// TIA Portal project "Lab3 with HMI" (V18)

(* hardware
DEVICE "HMI_1"  KTP700 Basic PN
   slot 0: "HMI_1"  KTP700 Basic PN  6AV2 123-2GB03-0AX0  15.1.0.0
   slot 1: "HMI_RT_1"  KTP700 Basic PN  6AV2 123-2GB03-0AX0  15.1.0.0
   slot 5: "HMI_1.IE_CP_1"  PROFINET Interface  15.0.1.0
      slot 1: "PROFINET Interface_1"  PROFINET Interface
         slot 1: "Port_1"  Port
DEVICE "S7-1200 station_1"  S7-1200 Station
   slot 0: "Rack_0"  S7-1200 Rack  Rack  V1.0
   slot 1: "PLC_1"  CPU 1214C DC/DC/DC  6ES7 214-1AG40-0XB0  V4.5
   slot 3: "ADC"  AQ1 signal board  6ES7 232-4HA30-0XB0  V1.0
DEVICE "S7-1200 station_2"  S7-1200 Station
   slot 0: "Rack_0"  S7-1200 Rack  Rack  V1.0
   slot 1: "PLC_2"  CPU 1215C DC/DC/DC  6ES7 215-1AG40-0XB0  V4.5
DEVICE "HMI_2"  KTP700 Basic PN
   slot 0: "HMI_2"  KTP700 Basic PN  6AV2 123-2GB03-0AX0  15.1.0.0
   slot 1: "HMI_RT_2"  KTP700 Basic PN  6AV2 123-2GB03-0AX0  15.1.0.0
   slot 5: "HMI_2.IE_CP_1"  PROFINET Interface  15.0.1.0
      slot 1: "PROFINET Interface_1"  PROFINET Interface
         slot 1: "Port_1"  Port
*)

// ===== PLC "PLC_1"  CPU 1214C DC/DC/DC =====

VAR_GLOBAL   // PLC tag table "Default tag table"
   "Start" AT %I0.6 : Bool;
   "Stop" AT %I0.7 : Bool;
   "Heating_Valve_Output" AT %Q0.2 : Bool;
   "Vent_Valve_Output" AT %Q0.3 : Bool;
   "DAC_Output" AT %QW80 : Word;
   "ADC_Input" AT %IW64 : Word;   // input is 0-10V ( 0 - 27648)
   "potentiometer" AT %Q1.1 : Bool;
END_VAR

DATA_BLOCK "Control_DB"   // DB1
{ S7_Optimized_Access := 'TRUE' }
VERSION : 0.1
   VAR
      HMI_Stop : Bool;   // Start button in the HMI panel
      HMI_Start : Bool;   // Stop button in the HMI panel
      Start_Stop : Bool;
      Input_Digital : Int;   // digital value 0 -27648
      Input_Norm : Real;   // normalize to 0 - 1
      Input_Volt : Real;   // scale to 0 - 10V
      Input_Celsius : Real;   // scale to 0 - 100 Celsius
      Output_Digital : Int;   // write to output in range of 0 - 27648
      Output_Volt : Real;
      Heating_On_Status : Bool;   // Heating valve is on
      Heating_Off_Status : Bool;   // Heating valve is off
      Vent_Status : Bool;   // Vent valve is on
   END_VAR
BEGIN
END_DATA_BLOCK

ORGANIZATION_BLOCK "Start_Stop"   // OB1, LAD, ProgramCycle
TITLE = "Main Program Sweep (Cycle)"
{ S7_Optimized_Access := 'TRUE' }
VERSION : 0.1
   VAR_INPUT
      Initial_Call : Bool;   // Initial call of this OB
      Remanence : Bool;   // =True, if remanent data are available
   END_VAR
BEGIN

REGION Network 1: Start and stop operation
   // Start pushbutton is normally opne (NO) switch.
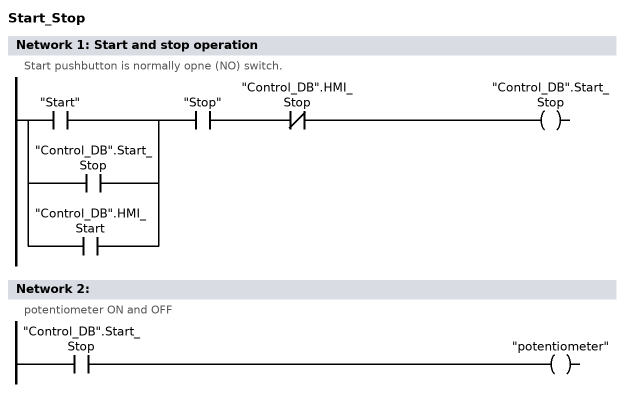
   RUNG wire#powerrail
      Contact( "Start" )
      wire#w1
      Contact( "Stop" )
      I_Contact( "Control_DB".HMI_Stop )
      Coil( "Control_DB".Start_Stop )
   END_RUNG
   RUNG wire#powerrail
      Contact( "Control_DB".Start_Stop )
   END_RUNG wire#w1
   RUNG wire#powerrail
      Contact( "Control_DB".HMI_Start )
   END_RUNG wire#w1
   // the same network as SCL:
   "Control_DB".Start_Stop := ("Start" OR "Control_DB".Start_Stop OR "Control_DB".HMI_Start) AND "Stop" AND NOT "Control_DB".HMI_Stop;
END_REGION

REGION Network 2
   // potentiometer ON and OFF
   RUNG wire#powerrail
      Contact( "Control_DB".Start_Stop )
      Coil( "potentiometer" )
   END_RUNG
   // the same network as SCL:
   "potentiometer" := "Control_DB".Start_Stop;
END_REGION
END_ORGANIZATION_BLOCK

ORGANIZATION_BLOCK "Controller"   // OB123, LAD, ProgramCycle
TITLE = "Main Program Sweep (Cycle)"
{ S7_Optimized_Access := 'TRUE' }
VERSION : 0.1
   VAR_INPUT
      Initial_Call : Bool;   // Initial call of this OB
      Remanence : Bool;   // =True, if remanent data are available
   END_VAR
BEGIN

REGION Network 1: Heating valve is on
   // Heating_ON_State is HIGH when temp less than 40 degree
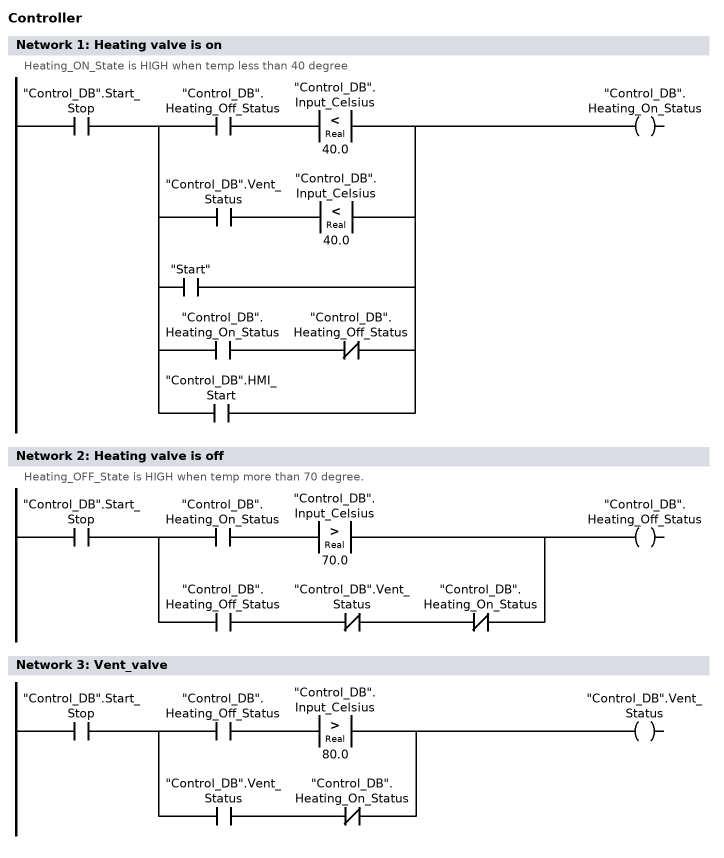
   RUNG wire#powerrail
      Contact( "Control_DB".Start_Stop )
      wire#w1
      Contact( "Control_DB".Heating_Off_Status )
      { S7_Templates := "SrcType := Real" } LT_Contact(in1 := "Control_DB".Input_Celsius, in2 := 40.0)
      wire#w2
      Coil( "Control_DB".Heating_On_Status )
   END_RUNG
   RUNG wire#w1
      Contact( "Control_DB".Vent_Status )
      { S7_Templates := "SrcType := Real" } LT_Contact(in1 := "Control_DB".Input_Celsius, in2 := 40.0)
   END_RUNG wire#w2
   RUNG wire#w1
      Contact( "Start" )
   END_RUNG wire#w2
   RUNG wire#w1
      Contact( "Control_DB".Heating_On_Status )
      I_Contact( "Control_DB".Heating_Off_Status )
   END_RUNG wire#w2
   RUNG wire#w1
      Contact( "Control_DB".HMI_Start )
   END_RUNG wire#w2
   // the same network as SCL:
   "Control_DB".Heating_On_Status := "Control_DB".Start_Stop AND (("Control_DB".Heating_Off_Status AND ("Control_DB".Input_Celsius < 40.0)) OR ("Control_DB".Vent_Status AND ("Control_DB".Input_Celsius < 40.0)) OR "Start" OR ("Control_DB".Heating_On_Status AND NOT "Control_DB".Heating_Off_Status) OR "Control_DB".HMI_Start);
END_REGION

REGION Network 2: Heating valve is off
   // Heating_OFF_State is HIGH when temp more than 70 degree.
   RUNG wire#powerrail
      Contact( "Control_DB".Start_Stop )
      wire#w1
      Contact( "Control_DB".Heating_On_Status )
      { S7_Templates := "SrcType := Real" } GT_Contact(in1 := "Control_DB".Input_Celsius, in2 := 70.0)
      wire#w2
      Coil( "Control_DB".Heating_Off_Status )
   END_RUNG
   RUNG wire#w1
      Contact( "Control_DB".Heating_Off_Status )
      I_Contact( "Control_DB".Vent_Status )
      I_Contact( "Control_DB".Heating_On_Status )
   END_RUNG wire#w2
   // the same network as SCL:
   "Control_DB".Heating_Off_Status := "Control_DB".Start_Stop AND (("Control_DB".Heating_On_Status AND ("Control_DB".Input_Celsius > 70.0)) OR ("Control_DB".Heating_Off_Status AND NOT "Control_DB".Vent_Status AND NOT "Control_DB".Heating_On_Status));
END_REGION

REGION Network 3: Vent_valve
   RUNG wire#powerrail
      Contact( "Control_DB".Start_Stop )
      wire#w1
      Contact( "Control_DB".Heating_Off_Status )
      { S7_Templates := "SrcType := Real" } GT_Contact(in1 := "Control_DB".Input_Celsius, in2 := 80.0)
      wire#w2
      Coil( "Control_DB".Vent_Status )
   END_RUNG
   RUNG wire#w1
      Contact( "Control_DB".Vent_Status )
      I_Contact( "Control_DB".Heating_On_Status )
   END_RUNG wire#w2
   // the same network as SCL:
   "Control_DB".Vent_Status := "Control_DB".Start_Stop AND (("Control_DB".Heating_Off_Status AND ("Control_DB".Input_Celsius > 80.0)) OR ("Control_DB".Vent_Status AND NOT "Control_DB".Heating_On_Status));
END_REGION
END_ORGANIZATION_BLOCK

ORGANIZATION_BLOCK "Temperature Sensor"   // OB124, LAD, ProgramCycle
TITLE = "Main Program Sweep (Cycle)"
{ S7_Optimized_Access := 'TRUE' }
VERSION : 0.1
   VAR_INPUT
      Initial_Call : Bool;   // Initial call of this OB
      Remanence : Bool;   // =True, if remanent data are available
   END_VAR
   VAR CONSTANT
      min : Int := 0;
      max : Int := 27648;
   END_VAR
BEGIN

REGION Network 1
   // copy the ADC to a Input_Digital variable
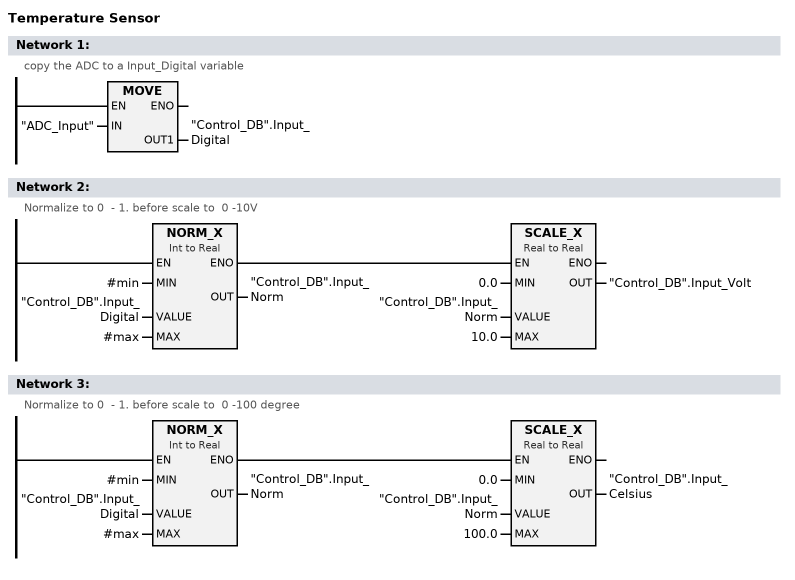
   RUNG wire#powerrail
      Move(in := "ADC_Input", out1 => "Control_DB".Input_Digital)
   END_RUNG
   // the same network as SCL:
   "Control_DB".Input_Digital := "ADC_Input";
END_REGION

REGION Network 2
   // Normalize to 0  - 1. before scale to  0 -10V
   RUNG wire#powerrail
      { S7_Templates := "[SrcType := Int, DestType := Real]" } Normalize(min := #min, value := "Control_DB".Input_Digital, max := #max, out => "Control_DB".Input_Norm)
      { S7_Templates := "[SrcType := Real, DestType := Real]" } Scale(min := 0.0, value := "Control_DB".Input_Norm, max := 10.0, out => "Control_DB".Input_Volt)
   END_RUNG
   // the same network as SCL:
   "Control_DB".Input_Norm := NORM_X(MIN := #min, VALUE := "Control_DB".Input_Digital, MAX := #max);
   "Control_DB".Input_Volt := SCALE_X(MIN := 0.0, VALUE := "Control_DB".Input_Norm, MAX := 10.0);
END_REGION

REGION Network 3
   // Normalize to 0  - 1. before scale to  0 -100 degree
   RUNG wire#powerrail
      { S7_Templates := "[SrcType := Int, DestType := Real]" } Normalize(min := #min, value := "Control_DB".Input_Digital, max := #max, out => "Control_DB".Input_Norm)
      { S7_Templates := "[SrcType := Real, DestType := Real]" } Scale(min := 0.0, value := "Control_DB".Input_Norm, max := 100.0, out => "Control_DB".Input_Celsius)
   END_RUNG
   // the same network as SCL:
   "Control_DB".Input_Norm := NORM_X(MIN := #min, VALUE := "Control_DB".Input_Digital, MAX := #max);
   "Control_DB".Input_Celsius := SCALE_X(MIN := 0.0, VALUE := "Control_DB".Input_Norm, MAX := 100.0);
END_REGION
END_ORGANIZATION_BLOCK

ORGANIZATION_BLOCK "Outputs"   // OB125, LAD, ProgramCycle
TITLE = "Main Program Sweep (Cycle)"
{ S7_Optimized_Access := 'TRUE' }
VERSION : 0.1
   VAR_INPUT
      Initial_Call : Bool;   // Initial call of this OB
      Remanence : Bool;   // =True, if remanent data are available
   END_VAR
BEGIN

REGION Network 1
   // A heating fluid control valve is open (valve open = TRUE)
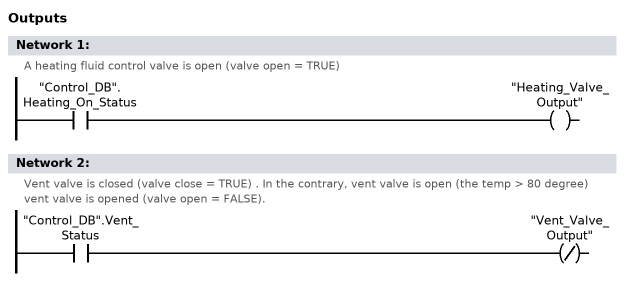
   RUNG wire#powerrail
      Contact( "Control_DB".Heating_On_Status )
      Coil( "Heating_Valve_Output" )
   END_RUNG
   // the same network as SCL:
   "Heating_Valve_Output" := "Control_DB".Heating_On_Status;
END_REGION

REGION Network 2
   // Vent valve is closed (valve close = TRUE) . In the contrary, vent valve is open (the temp > 80 degree) vent valve is opened (valve open = FALSE).
   RUNG wire#powerrail
      Contact( "Control_DB".Vent_Status )
      I_Coil( "Vent_Valve_Output" )
   END_RUNG
   // the same network as SCL:
   "Vent_Valve_Output" := NOT "Control_DB".Vent_Status;
END_REGION
END_ORGANIZATION_BLOCK

// ===== PLC "PLC_2"  CPU 1215C DC/DC/DC =====

VAR_GLOBAL   // PLC tag table "Default tag table"
   "Start" AT %I0.6 : Bool;
   "Stop" AT %I0.7 : Bool;
   "Heating_Valve_Output" AT %Q0.2 : Bool;
   "Vent_Valve_Output" AT %Q0.3 : Bool;
   "DAC_Output" AT %QW80 : Word;
   "ADC_Input" AT %IW64 : Word;
   "potentiometer" AT %Q1.1 : Bool;
END_VAR

DATA_BLOCK "Control_DB"   // DB1
{ S7_Optimized_Access := 'TRUE' }
VERSION : 0.1
   VAR
      HMI_Stop : Bool;   // Start button in the HMI panel
      HMI_Start : Bool;   // Stop button in the HMI panel
      Start_Stop : Bool;
      Input_Digital : Int;   // digital value 0 -27648
      Input_Norm : Real;   // normalize to 0 - 1
      Input_Volt : Real;   // scale to 0 - 10V
      Input_Celsius : Real;   // scale to 0 - 100 Celsius
      Output_Digital : Int;   // write to output in range of 0 - 27648
      Output_Volt : Real;
      Heating_On_Status : Bool;   // Heating valve is on
      Heating_Off_Status : Bool;   // Heating valve is off
      Vent_Status : Bool;   // Vent valve is on
   END_VAR
BEGIN
END_DATA_BLOCK

ORGANIZATION_BLOCK "Start_Stop"   // OB1, LAD, ProgramCycle
TITLE = "Main Program Sweep (Cycle)"
{ S7_Optimized_Access := 'TRUE' }
VERSION : 0.1
   VAR_INPUT
      Initial_Call : Bool;   // Initial call of this OB
      Remanence : Bool;   // =True, if remanent data are available
   END_VAR
BEGIN

REGION Network 1: Start and stop operation
   // Start pushbutton is normally opne (NO) switch.
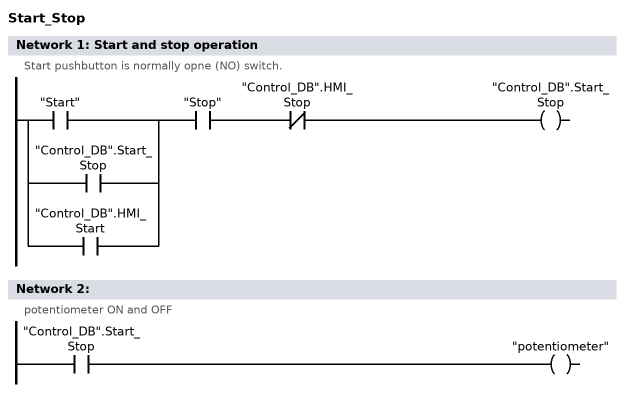
   RUNG wire#powerrail
      Contact( "Start" )
      wire#w1
      Contact( "Stop" )
      I_Contact( "Control_DB".HMI_Stop )
      Coil( "Control_DB".Start_Stop )
   END_RUNG
   RUNG wire#powerrail
      Contact( "Control_DB".Start_Stop )
   END_RUNG wire#w1
   RUNG wire#powerrail
      Contact( "Control_DB".HMI_Start )
   END_RUNG wire#w1
   // the same network as SCL:
   "Control_DB".Start_Stop := ("Start" OR "Control_DB".Start_Stop OR "Control_DB".HMI_Start) AND "Stop" AND NOT "Control_DB".HMI_Stop;
END_REGION

REGION Network 2
   // potentiometer ON and OFF
   RUNG wire#powerrail
      Contact( "Control_DB".Start_Stop )
      Coil( "potentiometer" )
   END_RUNG
   // the same network as SCL:
   "potentiometer" := "Control_DB".Start_Stop;
END_REGION
END_ORGANIZATION_BLOCK

ORGANIZATION_BLOCK "Controller"   // OB123, LAD, ProgramCycle
TITLE = "Main Program Sweep (Cycle)"
{ S7_Optimized_Access := 'TRUE' }
VERSION : 0.1
   VAR_INPUT
      Initial_Call : Bool;   // Initial call of this OB
      Remanence : Bool;   // =True, if remanent data are available
   END_VAR
BEGIN

REGION Network 1: Heating valve is on
   // Heating_ON_State is HIGH when temp less than 40 degree
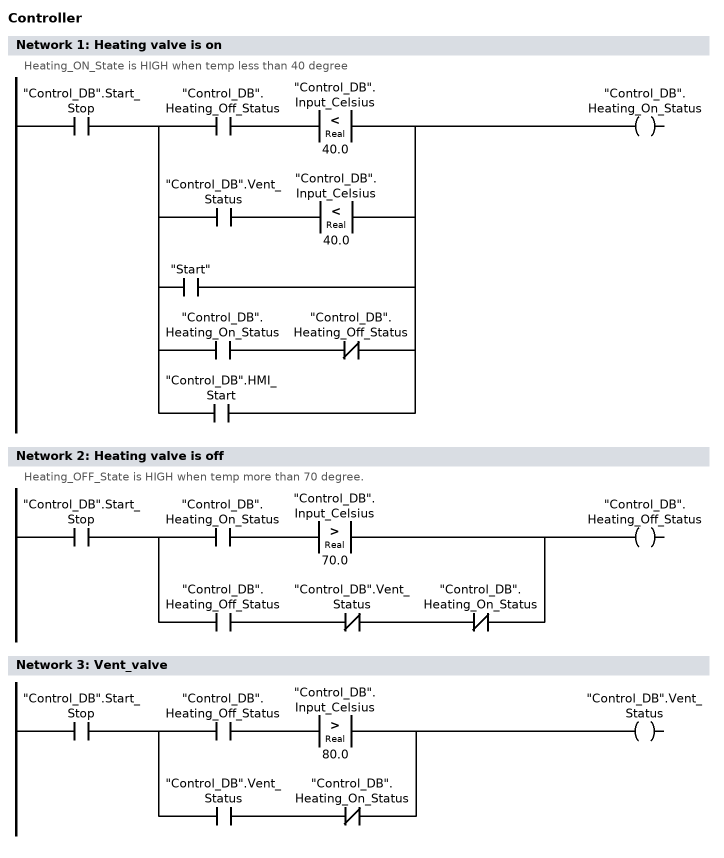
   RUNG wire#powerrail
      Contact( "Control_DB".Start_Stop )
      wire#w1
      Contact( "Control_DB".Heating_Off_Status )
      { S7_Templates := "SrcType := Real" } LT_Contact(in1 := "Control_DB".Input_Celsius, in2 := 40.0)
      wire#w2
      Coil( "Control_DB".Heating_On_Status )
   END_RUNG
   RUNG wire#w1
      Contact( "Control_DB".Vent_Status )
      { S7_Templates := "SrcType := Real" } LT_Contact(in1 := "Control_DB".Input_Celsius, in2 := 40.0)
   END_RUNG wire#w2
   RUNG wire#w1
      Contact( "Start" )
   END_RUNG wire#w2
   RUNG wire#w1
      Contact( "Control_DB".Heating_On_Status )
      I_Contact( "Control_DB".Heating_Off_Status )
   END_RUNG wire#w2
   RUNG wire#w1
      Contact( "Control_DB".HMI_Start )
   END_RUNG wire#w2
   // the same network as SCL:
   "Control_DB".Heating_On_Status := "Control_DB".Start_Stop AND (("Control_DB".Heating_Off_Status AND ("Control_DB".Input_Celsius < 40.0)) OR ("Control_DB".Vent_Status AND ("Control_DB".Input_Celsius < 40.0)) OR "Start" OR ("Control_DB".Heating_On_Status AND NOT "Control_DB".Heating_Off_Status) OR "Control_DB".HMI_Start);
END_REGION

REGION Network 2: Heating valve is off
   // Heating_OFF_State is HIGH when temp more than 70 degree.
   RUNG wire#powerrail
      Contact( "Control_DB".Start_Stop )
      wire#w1
      Contact( "Control_DB".Heating_On_Status )
      { S7_Templates := "SrcType := Real" } GT_Contact(in1 := "Control_DB".Input_Celsius, in2 := 70.0)
      wire#w2
      Coil( "Control_DB".Heating_Off_Status )
   END_RUNG
   RUNG wire#w1
      Contact( "Control_DB".Heating_Off_Status )
      I_Contact( "Control_DB".Vent_Status )
      I_Contact( "Control_DB".Heating_On_Status )
   END_RUNG wire#w2
   // the same network as SCL:
   "Control_DB".Heating_Off_Status := "Control_DB".Start_Stop AND (("Control_DB".Heating_On_Status AND ("Control_DB".Input_Celsius > 70.0)) OR ("Control_DB".Heating_Off_Status AND NOT "Control_DB".Vent_Status AND NOT "Control_DB".Heating_On_Status));
END_REGION

REGION Network 3: Vent_valve
   RUNG wire#powerrail
      Contact( "Control_DB".Start_Stop )
      wire#w1
      Contact( "Control_DB".Heating_Off_Status )
      { S7_Templates := "SrcType := Real" } GT_Contact(in1 := "Control_DB".Input_Celsius, in2 := 80.0)
      wire#w2
      Coil( "Control_DB".Vent_Status )
   END_RUNG
   RUNG wire#w1
      Contact( "Control_DB".Vent_Status )
      I_Contact( "Control_DB".Heating_On_Status )
   END_RUNG wire#w2
   // the same network as SCL:
   "Control_DB".Vent_Status := "Control_DB".Start_Stop AND (("Control_DB".Heating_Off_Status AND ("Control_DB".Input_Celsius > 80.0)) OR ("Control_DB".Vent_Status AND NOT "Control_DB".Heating_On_Status));
END_REGION
END_ORGANIZATION_BLOCK

ORGANIZATION_BLOCK "Temperature Sensor"   // OB124, LAD, ProgramCycle
TITLE = "Main Program Sweep (Cycle)"
{ S7_Optimized_Access := 'TRUE' }
VERSION : 0.1
   VAR_INPUT
      Initial_Call : Bool;   // Initial call of this OB
      Remanence : Bool;   // =True, if remanent data are available
   END_VAR
   VAR CONSTANT
      min : Int := 0;
      max : Int := 27648;
   END_VAR
BEGIN

REGION Network 1
   // copy the ADC to a Input_Digital variable
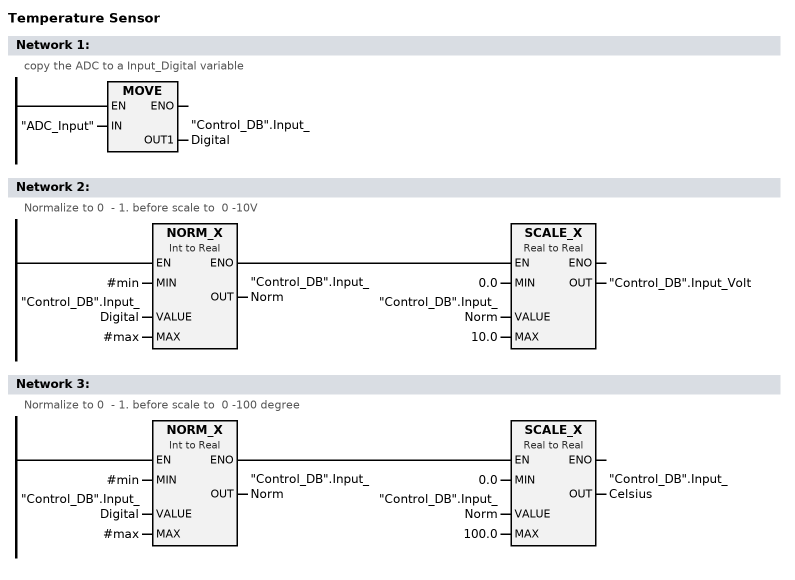
   RUNG wire#powerrail
      Move(in := "ADC_Input", out1 => "Control_DB".Input_Digital)
   END_RUNG
   // the same network as SCL:
   "Control_DB".Input_Digital := "ADC_Input";
END_REGION

REGION Network 2
   // Normalize to 0  - 1. before scale to  0 -10V
   RUNG wire#powerrail
      { S7_Templates := "[SrcType := Int, DestType := Real]" } Normalize(min := #min, value := "Control_DB".Input_Digital, max := #max, out => "Control_DB".Input_Norm)
      { S7_Templates := "[SrcType := Real, DestType := Real]" } Scale(min := 0.0, value := "Control_DB".Input_Norm, max := 10.0, out => "Control_DB".Input_Volt)
   END_RUNG
   // the same network as SCL:
   "Control_DB".Input_Norm := NORM_X(MIN := #min, VALUE := "Control_DB".Input_Digital, MAX := #max);
   "Control_DB".Input_Volt := SCALE_X(MIN := 0.0, VALUE := "Control_DB".Input_Norm, MAX := 10.0);
END_REGION

REGION Network 3
   // Normalize to 0  - 1. before scale to  0 -100 degree
   RUNG wire#powerrail
      { S7_Templates := "[SrcType := Int, DestType := Real]" } Normalize(min := #min, value := "Control_DB".Input_Digital, max := #max, out => "Control_DB".Input_Norm)
      { S7_Templates := "[SrcType := Real, DestType := Real]" } Scale(min := 0.0, value := "Control_DB".Input_Norm, max := 100.0, out => "Control_DB".Input_Celsius)
   END_RUNG
   // the same network as SCL:
   "Control_DB".Input_Norm := NORM_X(MIN := #min, VALUE := "Control_DB".Input_Digital, MAX := #max);
   "Control_DB".Input_Celsius := SCALE_X(MIN := 0.0, VALUE := "Control_DB".Input_Norm, MAX := 100.0);
END_REGION
END_ORGANIZATION_BLOCK

ORGANIZATION_BLOCK "Outputs"   // OB125, LAD, ProgramCycle
TITLE = "Main Program Sweep (Cycle)"
{ S7_Optimized_Access := 'TRUE' }
VERSION : 0.1
   VAR_INPUT
      Initial_Call : Bool;   // Initial call of this OB
      Remanence : Bool;   // =True, if remanent data are available
   END_VAR
BEGIN

REGION Network 1
   // A heating fluid control valve is open (valve open = TRUE)
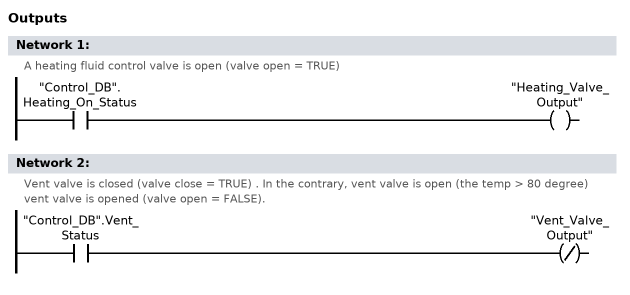
   RUNG wire#powerrail
      Contact( "Control_DB".Heating_On_Status )
      Coil( "Heating_Valve_Output" )
   END_RUNG
   // the same network as SCL:
   "Heating_Valve_Output" := "Control_DB".Heating_On_Status;
END_REGION

REGION Network 2
   // Vent valve is closed (valve close = TRUE) . In the contrary, vent valve is open (the temp > 80 degree) vent valve is opened (valve open = FALSE).
   RUNG wire#powerrail
      Contact( "Control_DB".Vent_Status )
      I_Coil( "Vent_Valve_Output" )
   END_RUNG
   // the same network as SCL:
   "Vent_Valve_Output" := NOT "Control_DB".Vent_Status;
END_REGION
END_ORGANIZATION_BLOCK

(* ===== HMI "HMI_RT_1" =====
system functions are stored by id; their names below are inferred from use
connection "HMI_Connection_1": ETHERNET, SMART_S7_1200_OMS

HMI tags "Default tag table"
   "Control_DB_HMI_Stop" : Bool = PLC Control_DB.HMI_Stop, 1 s
   "Control_DB_HMI_Start" : Bool = PLC Control_DB.HMI_Start AT %DB1.DBX0.0, 1 s
   "Control_DB_Start_Stop" : Bool = PLC Control_DB.Start_Stop AT %DB1.DBX0.0, 1 s
   "Control_DB_Heating_On_Status" : Bool = PLC Control_DB.Heating_On_Status AT %DB1.DBX0.0, 1 s
   "Control_DB_Input_Celsius" : Real = PLC Control_DB.Input_Celsius AT %DB1.DBX0.0, 1 s
   "Control_DB_Vent_Status" : Bool = PLC Control_DB.Vent_Status AT %DB1.DBD0, 1 s

screen "Root screen" 800x480, template "Template_1"
   Circle "Circle_1" at 319,94 size 40x40
      Appearance <- "Control_DB_Start_Stop"
   Button "Button_1" at 45,98 size 96x32; TextOff 'Start'
      on Press: SetBit("Control_DB_HMI_Start")
      on Release: ResetBit("Control_DB_HMI_Start")
   Button "Button_2" at 170,98 size 96x32; TextOff 'Stop'
      on Press: SetBit("Control_DB_HMI_Stop")
      on Release: ResetBit("Control_DB_HMI_Stop")
   Bar "Bar_1" at 603,64 size 119x372; MinimumValue 0; MaximumValue 100
      ProcessValue <- "Control_DB_Input_Celsius"
   TextField "Text field_1" at 91,338 size 43x23; Text 'Vent'
   Circle "Circle_2" at 207,210 size 48x48
      Appearance <- "Control_DB_Heating_On_Status"
   Circle "Circle_3" at 207,322 size 48x48
      Appearance <- "Control_DB_Vent_Status"
   TextField "Text field_2" at 92,225 size 69x23; Text 'Heating'
*)

(* ===== HMI "HMI_RT_2" =====
system functions are stored by id; their names below are inferred from use
connection "HMI_Connection_2": ETHERNET, SMART_S7_1200_OMS

HMI tags "Default tag table"
   "Control_DB_HMI_Start" : Bool = PLC Control_DB.HMI_Start, 1 s
   "Control_DB_Vent_Status" : Bool = PLC Control_DB.Vent_Status, 1 s
   "Control_DB_Heating_On_Status" : Bool = PLC Control_DB.Heating_On_Status, 1 s
   "Control_DB_Start_Stop" : Bool = PLC Control_DB.Start_Stop, 1 s
   "Control_DB_Input_Celsius" : Real = PLC Control_DB.Input_Celsius, 1 s
   "Control_DB_HMI_Stop" : Bool = PLC Control_DB.HMI_Stop, 1 s

screen "Root screen" 800x480, template "Template_1"
   Circle "Circle_1" at 319,94 size 40x40
      Appearance <- "Control_DB_Start_Stop"
   Button "Button_1" at 45,98 size 96x32; TextOff 'Start'
      on Release: ResetBit("Control_DB_HMI_Start")
      on Press: SetBit("Control_DB_HMI_Start")
   Button "Button_2" at 170,98 size 96x32; TextOff 'Stop'
      on Release: ResetBit("Control_DB_HMI_Stop")
      on Press: SetBit("Control_DB_HMI_Stop")
   Bar "Bar_1" at 603,64 size 119x372; MinimumValue 0; MaximumValue 100
      ProcessValue <- "Control_DB_Input_Celsius"
   TextField "Text field_1" at 91,338 size 43x23; Text 'Vent'
   Circle "Circle_2" at 207,210 size 48x48
      Appearance <- "Control_DB_Heating_On_Status"
   Circle "Circle_3" at 207,322 size 48x48
      Appearance <- "Control_DB_Vent_Status"
   TextField "Text field_2" at 92,225 size 69x23; Text 'Heating'
*)